{attribute 'linkalways'} 
{attribute 'no_explicit_call' := 'This FB is a CLASS and must be accessed using methods or properties'}
{attribute 'enable_dynamic_creation'}
FUNCTION_BLOCK SynchronousRpcResponse IMPLEMENTS I_SynchronousRpcResponse
VAR
	serverResponse : I_ServerResponse;
	serializer : I_Serializer;
	asynchronousRpcResponseFactory : I_AsynchronousRpcResponseFactory;
END_VAR

METHOD PUBLIC CompleteWithBase64
VAR_INPUT
	pBytes : POINTER TO BYTE;
	nBytes : DINT;
END_VAR
serializer.Reset();
serializer.AddBase64(pBytes, nBytes);
SendSuccessResponseUsingSeralizer(serializer);
END_METHOD

METHOD PUBLIC CompleteWithBool
VAR_INPUT
	Value : BOOL;
END_VAR
serializer.Reset();
serializer.AddBool(Value);
SendSuccessResponseUsingSeralizer(serializer);
END_METHOD

METHOD PUBLIC CompleteWithBytesAsHex
VAR_INPUT
	pBytes : POINTER TO BYTE;
	nBytes : DINT;
END_VAR
serializer.Reset();
serializer.AddBytesAsHex(pBytes, nBytes);
SendSuccessResponseUsingSeralizer(serializer);
END_METHOD

METHOD PUBLIC CompleteWithDateTime
VAR_INPUT
	Value : DATE_AND_TIME;
END_VAR
serializer.Reset();
serializer.AddDateTime(Value);
SendSuccessResponseUsingSeralizer(serializer);
END_METHOD

METHOD PUBLIC CompleteWithDcTime
VAR_INPUT
	Value : DCTIME;
END_VAR
serializer.Reset();
serializer.AddDcTime(Value);
SendSuccessResponseUsingSeralizer(serializer);
END_METHOD

METHOD PUBLIC CompleteWithDint
VAR_INPUT
	Value : DINT;
END_VAR
serializer.Reset();
serializer.AddDint(Value);
SendSuccessResponseUsingSeralizer(serializer);
END_METHOD

METHOD PUBLIC CompleteWithFileTime
VAR_INPUT
	Value : FILETIME;
END_VAR
serializer.Reset();
serializer.AddFileTime(Value);
SendSuccessResponseUsingSeralizer(serializer);
END_METHOD

METHOD PUBLIC CompleteWithLint
VAR_INPUT
	Value : LINT;
END_VAR
serializer.Reset();
serializer.AddLint(Value);
SendSuccessResponseUsingSeralizer(serializer);
END_METHOD

METHOD PUBLIC CompleteWithLreal
VAR_INPUT
	Value : LREAL;
END_VAR
serializer.Reset();
serializer.AddLreal(Value);
SendSuccessResponseUsingSeralizer(serializer);
END_METHOD

METHOD PUBLIC CompleteWithNull
VAR_INPUT
END_VAR
serializer.Reset();
serializer.AddNull();
SendSuccessResponseUsingSeralizer(serializer);
END_METHOD

METHOD PUBLIC CompleteWithObject
VAR_INPUT
	Object : I_Serializable;
END_VAR
serializer.Reset();
Object.SerializeWith(serializer);
SendSuccessResponseUsingSeralizer(serializer);
END_METHOD

METHOD PUBLIC CompleteWithReal
VAR_INPUT
	Value : REAL;
END_VAR
serializer.Reset();
serializer.AddReal(Value);
SendSuccessResponseUsingSeralizer(serializer);
END_METHOD

METHOD PUBLIC CompleteWithSerializer
VAR_INPUT
	Serializer : I_Serializer;
END_VAR
SendSuccessResponseUsingSeralizer(Serializer);
END_METHOD

METHOD PUBLIC CompleteWithString
VAR_INPUT
	Value : T_MAXSTRING;
END_VAR
serializer.Reset();
serializer.AddString(Value);
SendSuccessResponseUsingSeralizer(serializer);
END_METHOD

METHOD PUBLIC CompleteWithUdint
VAR_INPUT
	Value : UDINT;
END_VAR
serializer.Reset();
serializer.AddUdint(Value);
SendSuccessResponseUsingSeralizer(serializer);
END_METHOD

METHOD PUBLIC CompleteWithUlint
VAR_INPUT
	Value : ULINT;
END_VAR
serializer.Reset();
serializer.AddUlint(Value);
SendSuccessResponseUsingSeralizer(serializer);
END_METHOD

METHOD FB_exit : BOOL
VAR_INPUT
	bInCopyCode : BOOL; // if TRUE, the exit method is called for exiting an instance that is copied afterwards (online change).
END_VAR
IF bInCopyCode THEN
	RETURN;
END_IF

serializer.Dispose();
END_METHOD

METHOD FB_init : BOOL
VAR_INPUT
	bInitRetains : BOOL; // if TRUE, the retain variables are initialized (warm start / cold start)
	bInCopyCode : BOOL;  // if TRUE, the instance afterwards gets moved into the copy code (online change)
	ServerResponse : I_ServerResponse;
	Serializer : I_Serializer;
	AsynchronousRpcResponseFactory : I_AsynchronousRpcResponseFactory;
END_VAR
THIS^.serverResponse := ServerResponse;
THIS^.serializer := Serializer.Clone();
THIS^.asynchronousRpcResponseFactory := AsynchronousRpcResponseFactory;
END_METHOD

METHOD PUBLIC GetSerializer : I_Serializer
VAR_INPUT
END_VAR
GetSerializer := serializer.Clone();
END_METHOD

METHOD PUBLIC RejectWithMessage
VAR_INPUT
	Message : T_MAXSTRING;
END_VAR
serverResponse.Error(Message);
END_METHOD

METHOD PROTECTED SendSuccessResponseUsingSeralizer
VAR_INPUT
	Serializer : I_Serializer;
END_VAR
VAR
	jsonSize : UDINT;
	pJsonString : POINTER TO STRING;
END_VAR
jsonSize := Serializer.GetSeralizedDataLength();

IF jsonSize = 0 THEN
	serverResponse.Success();
END_IF

pJsonString := __NEW(BYTE, jsonSize);

IF NOT Serializer.TryGetSerialziedData(pJsonString, jsonSize) THEN
	serverResponse.Error('RPC Handler unable to get serialized data');
	__DELETE(pJsonString);
	RETURN;
END_IF

serverResponse.SuccessWithPayload(pJsonString, jsonSize);
__DELETE(pJsonString);
END_METHOD

METHOD PUBLIC TryMakeAsynchronous : BOOL
VAR_INPUT
	Destination : REFERENCE TO I_AsynchronousRpcResponse;
END_VAR
TryMakeAsynchronous := asynchronousRpcResponseFactory.TryCreate(Destination);
END_METHOD

END_FUNCTION_BLOCK

(* stored: Version 1.1.0.1, ProductVersion 3.1.4024.12
   POU SynchronousRpcResponse: Id {c724498f-baf7-4f00-9137-6c3a66aa5cd0}, SpecialFunc None
   Folder Constructor: Id {12740898-8cc4-4e25-8ce9-9fc0666115c8}
   Folder Destructor: Id {c48347be-f693-4190-9e96-0dd879b63060}
   Folder Protected: Id {dcb37f09-2ecb-4483-9579-8dcbc7918f05}
   Method CompleteWithBase64: Id {1852c73b-7584-42d8-8595-d755b4b78f03}
   Method CompleteWithBool: Id {7e7403d7-f4cb-400d-8ab9-ff3aedbf57b4}
   Method CompleteWithBytesAsHex: Id {93903bbf-3c38-4980-8b1f-e2263cdb86e0}
   Method CompleteWithDateTime: Id {20014026-b2b6-43a2-93d7-0a69b7b874c8}
   Method CompleteWithDcTime: Id {601da881-ce92-48c2-b16a-901c433dac2e}
   Method CompleteWithDint: Id {38773dc1-5afc-4fbe-8d85-19dcb6f6dec0}
   Method CompleteWithFileTime: Id {ce3c3570-3dbd-429b-a0df-6122eef0b941}
   Method CompleteWithLint: Id {15fb45be-f8cd-476e-936e-95dd739d2ad8}
   Method CompleteWithLreal: Id {a6f94923-7cc9-4772-9c0b-daa067666dd8}
   Method CompleteWithNull: Id {a26a3275-f5d8-4d82-a9fa-28465a681661}
   Method CompleteWithObject: Id {8c148a58-c3ff-4c45-bfcd-db6bebceaad0}
   Method CompleteWithReal: Id {c45e6c4a-0553-4bd2-a3cd-0a5b5bd48d1b}
   Method CompleteWithSerializer: Id {10656fd7-dd8c-4e2c-a443-082c5750c598}
   Method CompleteWithString: Id {abf0072f-fd49-4976-9966-a04a5b803fee}
   Method CompleteWithUdint: Id {859ce20a-da2e-47f5-ba72-c20e7d8c636d}
   Method CompleteWithUlint: Id {c6871ed5-3419-4e00-9dd1-9901890cf472}
   Method FB_exit: Id {a21d938a-cfc7-4b8d-a8b3-12edc530b065}
   Method FB_init: Id {58740322-7d24-44d6-95e0-bd81b1ebde4a}
   Method GetSerializer: Id {3c95a31f-9472-4fa2-8b38-a78edbb5c949}
   Method RejectWithMessage: Id {d016a36c-5bb1-48bd-ab36-b1534a482e0e}
   Method SendSuccessResponseUsingSeralizer: Id {e0fd64b5-8f20-4205-b67f-95b2daa27c70}
   Method TryMakeAsynchronous: Id {e3d7ce72-9753-4130-a9b0-5dfe11ab3e76} *)
